FUNCTION_BLOCK AutoSamplar_Manager (* Basic Function Block Type *)
  (* Standard: 61499-2 *)
  (* Version 0.0, 9/26/2024, SESA713705, Schneider Electric, Template *)
  PACKAGE SE.Nereda;
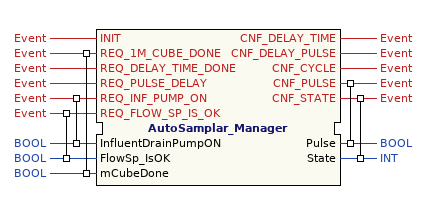
  EVENT_INPUT
    INIT;
    REQ_1M_CUBE_DONE WITH mCubeDone;
    REQ_DELAY_TIME_DONE;
    REQ_PULSE_DELAY;
    REQ_INF_PUMP_ON WITH InfluentDrainPumpON;
    REQ_FLOW_SP_IS_OK WITH FlowSp_IsOK;
  END_EVENT
  EVENT_OUTPUT
    CNF_DELAY_TIME;
    CNF_DELAY_PULSE;
    CNF_CYCLE;
    CNF_PULSE WITH Pulse;
    CNF_STATE WITH State;
  END_EVENT
  VAR_INPUT
    InfluentDrainPumpON : BOOL;
    FlowSp_IsOK : BOOL;
    mCubeDone : BOOL;
  END_VAR
  VAR_OUTPUT
    Pulse : BOOL;
    State : INT;
  END_VAR
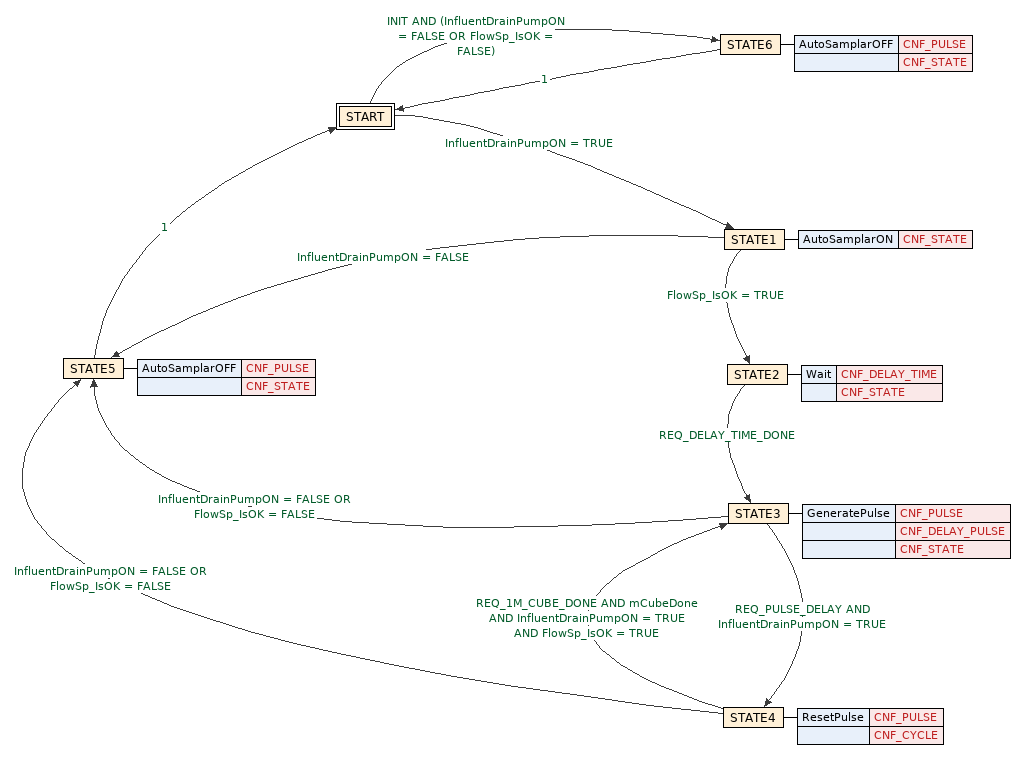
  EC_STATES
    START; (* Initial State *)
    STATE1 : AutoSamplarON -> CNF_STATE;
    STATE2 : Wait -> CNF_DELAY_TIME, -> CNF_STATE;
    STATE3 : GeneratePulse -> CNF_PULSE, -> CNF_DELAY_PULSE, -> CNF_STATE;
    STATE4 : ResetPulse -> CNF_PULSE, -> CNF_CYCLE;
    STATE5 : AutoSamplarOFF -> CNF_PULSE, -> CNF_STATE;
    STATE6 : AutoSamplarOFF -> CNF_PULSE, -> CNF_STATE;
  END_STATES
  EC_TRANSITIONS
    START TO STATE1 := InfluentDrainPumpON = TRUE;
    STATE1 TO STATE2 := FlowSp_IsOK = TRUE;
    STATE2 TO STATE3 := REQ_DELAY_TIME_DONE;
    STATE3 TO STATE4 := REQ_PULSE_DELAY AND InfluentDrainPumpON = TRUE;
    STATE4 TO STATE3 := REQ_1M_CUBE_DONE AND mCubeDone AND InfluentDrainPumpON = TRUE AND FlowSp_IsOK = TRUE;
    STATE3 TO STATE5 := InfluentDrainPumpON = FALSE OR FlowSp_IsOK = FALSE;
    STATE4 TO STATE5 := InfluentDrainPumpON = FALSE OR FlowSp_IsOK = FALSE;
    STATE5 TO START := 1;
    START TO STATE6 := INIT AND (InfluentDrainPumpON = FALSE OR FlowSp_IsOK = FALSE);
    STATE6 TO START := 1;
    STATE1 TO STATE5 := InfluentDrainPumpON = FALSE;
  END_TRANSITIONS
  ALGORITHM AutoSamplarON IN ST:
;
State := 1;
  END_ALGORITHM
  ALGORITHM GeneratePulse IN ST:
;
Pulse := TRUE;
State := 3;
  END_ALGORITHM
  ALGORITHM ResetPulse IN ST:
;
Pulse := FALSE;
  END_ALGORITHM
  ALGORITHM AutoSamplarOFF IN ST:
;
Pulse := FALSE;
State := 0;
  END_ALGORITHM
  ALGORITHM Wait IN ST:
;
State := 2;
  END_ALGORITHM
END_FUNCTION_BLOCK
